TYPE Status_Waegesystem : (Kalibrieren, Wiegen);
END_TYPE

(* stored: Version 1.1.0.1, ProductVersion 3.1.4019.2
   DUT Status_Waegesystem: Id {6662074b-1010-48ce-8355-27be617da273} *)
